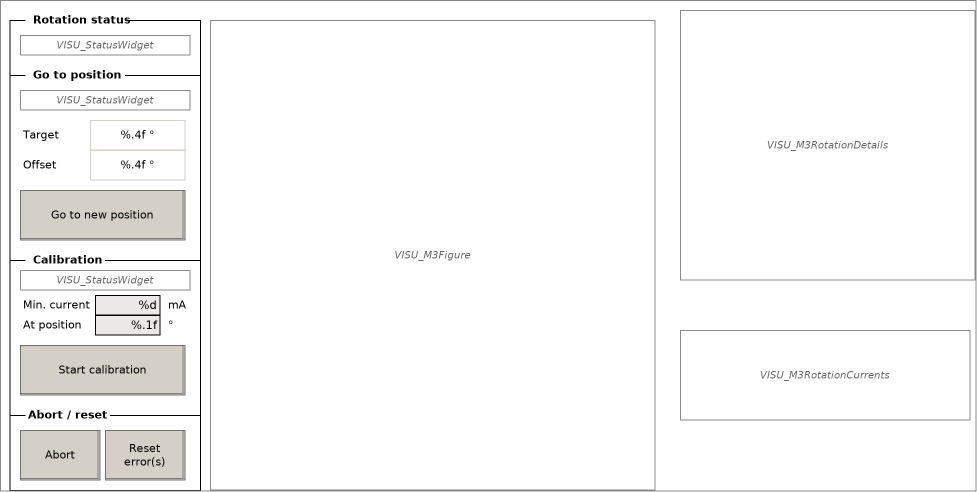
VISUALIZATION VISU_M3Rotation_General  // 977x492
VAR_IN_OUT
	ref : M3Rotation;
    widget : M3RotationWidget;
    m3Ref : M3;
    m3Widget : M3Widget;
END_VAR
    Button (20,190 165x50), "Go to new position", input disabled if: ref.processes.goto.statuses.enabledStatus.disabled
        OnMouseClick: execute { ref.processes.goto.do_request := TRUE; }
    Frame (210,20 445x470)
        shows VISU_M3Figure(m3 := m3Ref, widget := m3Widget, hideDetails := m3Widget.NO)
    Textfield (90,120 95x30), "%.4f °", text variable: ref.processes.goto.set.position
        OnMouseClick: write the text variable via Default
    Label (20,120 70x30), "Target"
    Label (20,150 70x30), "Offset"
    Textfield (90,150 95x30), "%.4f °", text variable: ref.processes.goto.set.offset
        OnMouseClick: write the text variable via Default
    Button (20,430 80x50), "Abort", input disabled if: ref.processes.abort.statuses.enabledStatus.disabled
        OnMouseClick: execute { ref.processes.abort.do_request := TRUE; }
    Frame (680,10 295x270)
        shows VISU_M3RotationDetails(ref := ref, widget := widget)
    Label (30,60 150x30), "Go to position"
    Line (125,75) (200,75)
    Line (10,75) (25,75)
    Line (200,20) (200,490)
    Frame (20,90 170x20)
        shows VISU_StatusWidget(widget := widget.gotoProcedureStatus)
    Button (105,430 80x50), "Reset error(s)", input disabled if: ref.processes.reset.statuses.enabledStatus.disabled
        OnMouseClick: execute { ref.processes.reset.do_request := TRUE; }
    Label (30,5 150x30), "Rotation status"
    Line (125,20) (200,20)
    Line (10,20) (25,20)
    Frame (20,35 170x20)
        shows VISU_StatusWidget(widget := widget.actualStatus)
    Line (105,260) (200,260)
    Label (30,245 75x30), "Calibration"
    Line (10,260) (25,260)
    Frame (20,270 170x20)
        shows VISU_StatusWidget(widget := widget.calibrateProcedureStatus)
    Button (20,345 165x50), "Start calibration", input disabled if: ref.processes.calibrate.statuses.enabledStatus.disabled
        OnMouseClick: execute { ref.processes.calibrate.do_request := TRUE; }
    Line (10,490) (200,490)
    Label (20,295 100x20), "Min. current"
    Label (165,295 35x20), "mA"
    Rectangle (95,295 65x20), "%d", text variable: ref.parts.calibrateProcedure.minimumCurrent
    Rectangle (95,315 65x20), "%.1f", text variable: ref.parts.calibrateProcedure.minimumCurrentPosition
    Label (165,315 35x20), "°"
    Label (20,315 70x20), "At position"
    Line (10,490) (10,20)
    Line (110,415) (200,415)
    Label (25,400 85x30), "Abort / reset"
    Line (10,415) (25,415)
    Frame (680,330 290x90)
        shows VISU_M3RotationCurrents(ref := ref, widget := widget)
END_VISUALIZATION

(* stored: Version 1.1.0.1, ProductVersion 3.1.4019.2
   Visu VISU_M3Rotation_General: Id {4773f1e1-4fb9-4392-aee6-4038f38532c1} *)
